Staubli VAL3: Endlosschleife.pjx

--- Endlosschleife.pjx ---
Parameters version=s7.5.3 stackSize=5000 millimeterUnit=true
Program file=MoveJoint.pgx
Program file=MoveLine.pgx
Program file=start.pgx
Program file=stop.pgx
Program file=main.pgx
Data file=Endlosschleife.dtx

--- main.pgx ---
program main()
begin
    pPointRx1.config.shoulder = lefty
    pPointRx1.config.elbow = epositive
    pPointRx1.config.wrist = wpositive
    pPointRx2.config.shoulder = lefty
    pPointRx2.config.elbow = epositive
    pPointRx2.config.wrist = wpositive
    mCurrentSpeed.tvel = 100.00
    mCurrentSpeed.blend = joint
    mCurrentSpeed.reach = 0.010
    mCurrentSpeed.leave = 0.010
    		// Program Endlosschleife start
		// Program generated by RoboDK v5.2.1 for Staubli TX2-40 on 26/04/2021 14:06:26
		link(pPointRx1,StaubliTX240Base)
		link(pPointRx2,StaubliTX240Base)
		call MoveJoint(0.00000,0.00000,90.00000,0.00000,0.00000,-0.00000)
		while true
			call MoveJoint(0.75339,44.25550,52.41940,0.00000,83.32510,0.75339)
			call MoveJoint(-10.97790,47.35230,41.99440,0.00000,90.65320,-10.97790)
			call MoveJoint(-1.36528,60.04990,34.36770,0.00000,85.58250,-1.36528)
			call MoveJoint(0.00000,0.00000,90.00000,0.00000,0.00000,-0.00000)
		endWhile

		waitEndMove()
		// Program Endlosschleife end

end
